TYPE ST_AxisInputs :
STRUCT
    bLimitFwd AT %I*: BOOL;
    bLimitBwd AT %I*: BOOL;
    bHomeSensor AT %I*: BOOL; //Reference siganl for homing
END_STRUCT
END_TYPE

(* stored: Version 1.1.0.1, ProductVersion 3.1.4024.5
   DUT ST_AxisInputs: Id {c688a7fd-4b78-4e23-92c9-09a1ce1d0174} *)
